INTERFACE ITF_SITP_Element

(*			
	EVERDE sp. z o.o.
	Rafał Osajda		25.02.2025		TC 4026.13		wer. 0.0.0.1
	Aktualizuje czas pracy w stanie
*)
METHOD PUBLIC AktualizujCzas
VAR_INPUT
	tInterwal			: time;
END_VAR
END_METHOD

METHOD PUBLIC ustawAktywny
VAR_INPUT
	bIN		: BOOL;
END_VAR
END_METHOD

METHOD PUBLIC UstawNazwe
VAR_INPUT
	stNazwa					: B_Baza.ST_Etykieta;
END_VAR
END_METHOD

METHOD PUBLIC ustawWlaczony
VAR_INPUT
	bIN		: bool;
END_VAR
END_METHOD

METHOD PUBLIC WywolajAkcjePBDlaStanu : BOOL
VAR_INPUT
	iNumerPB				: INT;
END_VAR
END_METHOD

(*			
	EVERDE sp. z o.o.
	Rafał Osajda		25.02.2025		TC 4026.13		wer. 0.0.0.1
	Zeruje wartość czasu
*)
METHOD PUBLIC ZerujCzas
VAR_INPUT
END_VAR
END_METHOD

METHOD zwrocAktywny : BOOL
VAR_INPUT
END_VAR
END_METHOD

METHOD PUBLIC zwrocCzas : STRING
VAR_INPUT
END_VAR
END_METHOD

(*			
	EVERDE sp. z o.o.
	Rafał Osajda		18.06.2025		TC 4024.66
	Zwraca true jak wyjście ze stanu jest możliwe
*)
METHOD PUBLIC ZwrocCzyMoznaWyjscZeStanu : BOOL
END_METHOD

METHOD PUBLIC zwrocLCzas : LTIME
VAR_INPUT
END_VAR
END_METHOD

METHOD PUBLIC ZwrocNazwe : WSTRING
VAR_INPUT
END_VAR
END_METHOD

METHOD PUBLIC zwrocWlaczony : BOOL
VAR_INPUT
END_VAR
END_METHOD

END_INTERFACE

(* stored: Version 1.1.0.1
   Itf ITF_SITP_Element: Id {56ad140b-2e24-0456-2903-45f6811caf3f}
   Method AktualizujCzas: Id {9fddaafb-4935-0cd6-10a2-41e053f34a97}
   Method ustawAktywny: Id {83d90448-4feb-0931-1ce5-5f783a323b55}
   Method UstawNazwe: Id {30c6e5a8-7d3c-0879-0e59-6555b74b7c14}
   Method ustawWlaczony: Id {e6958d95-2f38-0d32-1750-ed5c61d2d219}
   Method WywolajAkcjePBDlaStanu: Id {d4f9ec06-7eac-0d01-3680-76f435d6632e}
   Method ZerujCzas: Id {d9c7d326-1031-0e68-11eb-311b63586d82}
   Method zwrocAktywny: Id {760299c5-415b-0a5a-0458-7bce8628bdba}
   Method zwrocCzas: Id {0e8791cb-23c0-0a2c-2cd6-6de8360dcdc4}
   Method ZwrocCzyMoznaWyjscZeStanu: Id {47bb149c-6b91-0a3d-0cd3-620c340ce16a}
   Method zwrocLCzas: Id {aa91922f-d5b5-04ad-2346-7642373f3b16}
   Method ZwrocNazwe: Id {40319fda-86a3-0baa-1c6d-71cf675a5258}
   Method zwrocWlaczony: Id {49bf9efa-05da-07d2-20ae-eaba0b2065bf} *)
